// Mitsubishi GX Works2 project: Class4_Traffic Lights   PLC: Q03UD

PROGRAM MAIN
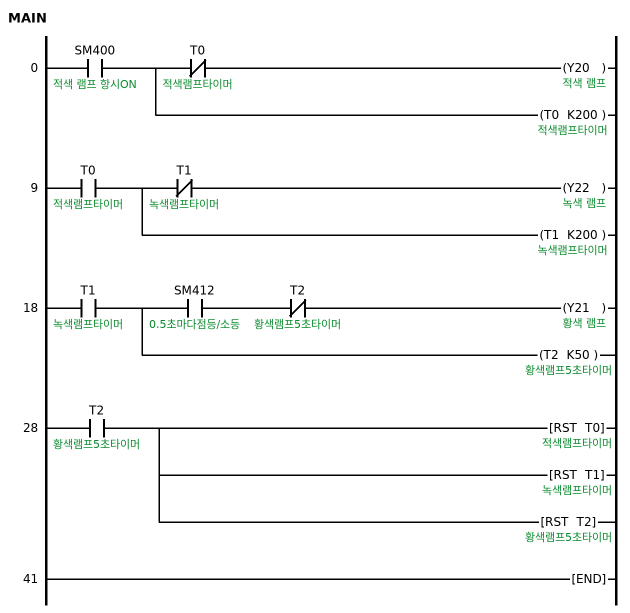
0     LD      SM400  ; 적색 램프 항시ON
      MPS
      ANI     T0  ; 적색램프타이머
      OUT     Y20  ; 적색 램프
      MPP
      OUT     T0 K200  ; 적색램프타이머
9     LD      T0  ; 적색램프타이머
      MPS
      ANI     T1  ; 녹색램프타이머
      OUT     Y22  ; 녹색 램프
      MPP
      OUT     T1 K200  ; 녹색램프타이머
18    LD      T1  ; 녹색램프타이머
      MPS
      AND     SM412  ; 0.5초마다점등/소등
      ANI     T2  ; 황색램프5초타이머
      OUT     Y21  ; 황색 램프
      MPP
      OUT     T2 K50  ; 황색램프5초타이머
28    LD      T2  ; 황색램프5초타이머
      RST     T0  ; 적색램프타이머
      RST     T1  ; 녹색램프타이머
      RST     T2  ; 황색램프5초타이머
41    END
END_PROGRAM

// device comments not shown above
M0  ; 빨간램프 스위치
M1  ; 노란램프 스위치
M2  ; 녹색램프 스위치
D0  ; 리셋
